# EPICS autosave request: ESP300/iocBoot/ioc_esp_bmb/auto_positions.req
file "XFM_motor_positions.req",      P=XF:04BMB-OP:, M=MBV-Cam:Y:Mtr
